(* Schneider Machine Expert - Basic project control, file version 2.9.0.0 *)
(* ProjectInformations: Name=Nuevo proyecto *)

HARDWARE
  Cpu 0: TM221M16R/G
  EthernetConfiguration: NetworkName=M221, IpAllocationMode=FixedAddress, IpAddress=0.0.0.0, SubnetMask=0.0.0.0
  SerialLineConfiguration: Baud=Baud19200, Parity=ParityEven, DataBits=DataBits8, StopBits=StopBits1, PhysicalMedium=PhysicalMediumRs485, TransmissionMode=TransmissionModeModbusRtu, SlaveId=1, Addressing=SlaveAddressing
  MastTask: UsePeriodScanMode=true, PeriodScan=10
  FastTask: Period=255
  CpuBehavior: StartingMode=StartAsPreviousState, AutoSaveRamOnEeprom=true, WatchdogPeriod=250

SYMBOLS  (address, symbol, comment, settings)
  %MW500    ERR
  %MW501    VEL
  %MW502    THETA
  %MW503    CRISP
  %MF1      REAL_ERROR
  %MF10     ENL
  %MF19     ENM
  %MF28     ENP
  %MF37     EZ
  %MF46     EPP
  %MF55     EPM
  %MF64     EPL
  %MF67     REAL_VEL
  %MF76     VNL
  %MF85     VNM
  %MF94     VNP
  %MF103    VZ
  %MF112    VPP
  %MF121    VPM
  %MF130    VPL
  %MF133    REAL_THETA
  %MF142    NL
  %MF151    NM
  %MF160    Z
  %MF169    PM
  %MF178    PL
  %MF181    W1
  %MF184    W2
  %MF187    W3
  %MF190    W4
  %MF193    W5
  %MF196    W6
  %MF199    W7
  %MF202    W8
  %MF205    W9
  %MF208    W10
  %MF211    W11
  %MF214    W12
  %MF217    W13
  %MF220    W14
  %MF223    W15
  %MF226    W16
  %MF229    W17
  %MF232    W18
  %MF235    W19
  %MF238    W20
  %MF241    W21
  %MF244    W22
  %MF247    W23
  %MF250    W24
  %MF253    W25
  %MF283    NUM
  %MF301    DEN

POU Nuevo POU
  (* SectionNumber=1 *)

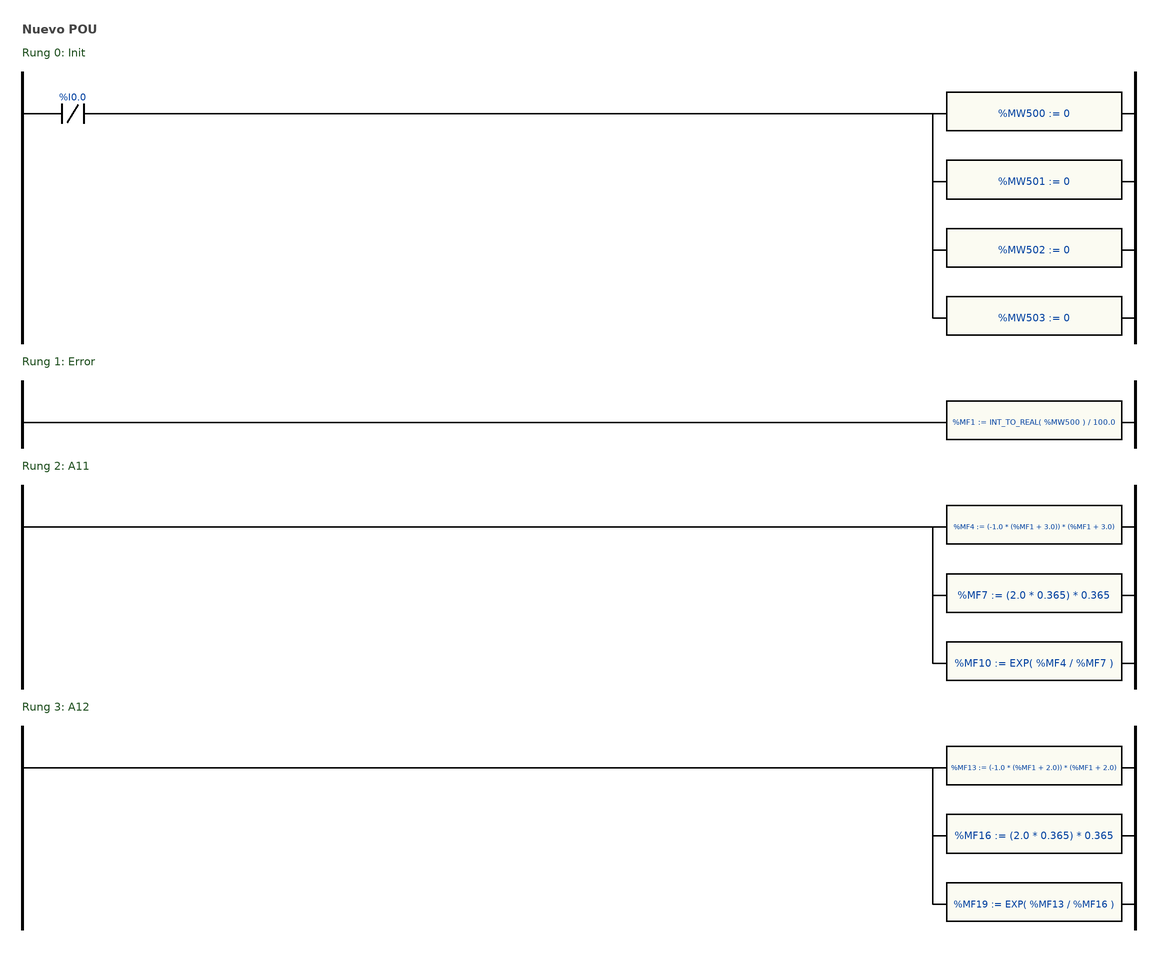

// Rung 0: Init
  LDN %I0.0
  [ %MW500 := 0 ]         (* ERR *)
  [ %MW501 := 0 ]         (* VEL *)
  [ %MW502 := 0 ]         (* THETA *)
  [ %MW503 := 0 ]         (* CRISP *)
  // as ST:
  //   IF NOT %I0.0 THEN ERR := 0; END_IF;
  //   IF NOT %I0.0 THEN VEL := 0; END_IF;
  //   IF NOT %I0.0 THEN THETA := 0; END_IF;
  //   IF NOT %I0.0 THEN CRISP := 0; END_IF;

// Rung 1: Error
  LD 1
  [ %MF1 := INT_TO_REAL ( %MW500 ) / 100.0 ](* REAL_ERROR, ERR *)
  // as ST:
  //   REAL_ERROR := INT_TO_REAL ( ERR ) / 100.0;

// Rung 2: A11
  LD 1
  [ %MF4 := ( -1.0 * ( %MF1 + 3.0 ) ) * ( %MF1 + 3.0 ) ](* REAL_ERROR, REAL_ERROR *)
  [ %MF7 := ( 2.0 * 0.365 ) * 0.365 ]
  [ %MF10 := EXP ( %MF4 / %MF7 ) ](* ENL *)
  // as ST:
  //   %MF4 := ( -1.0 * ( REAL_ERROR + 3.0 ) ) * ( REAL_ERROR + 3.0 );
  //   %MF7 := ( 2.0 * 0.365 ) * 0.365;
  //   ENL := EXP ( %MF4 / %MF7 );

// Rung 3: A12
  LD 1
  [ %MF13 := ( -1.0 * ( %MF1 + 2.0 ) ) * ( %MF1 + 2.0 ) ](* REAL_ERROR, REAL_ERROR *)
  [ %MF16 := ( 2.0 * 0.365 ) * 0.365 ]
  [ %MF19 := EXP ( %MF13 / %MF16 ) ](* ENM *)
  // as ST:
  //   %MF13 := ( -1.0 * ( REAL_ERROR + 2.0 ) ) * ( REAL_ERROR + 2.0 );
  //   %MF16 := ( 2.0 * 0.365 ) * 0.365;
  //   ENM := EXP ( %MF13 / %MF16 );

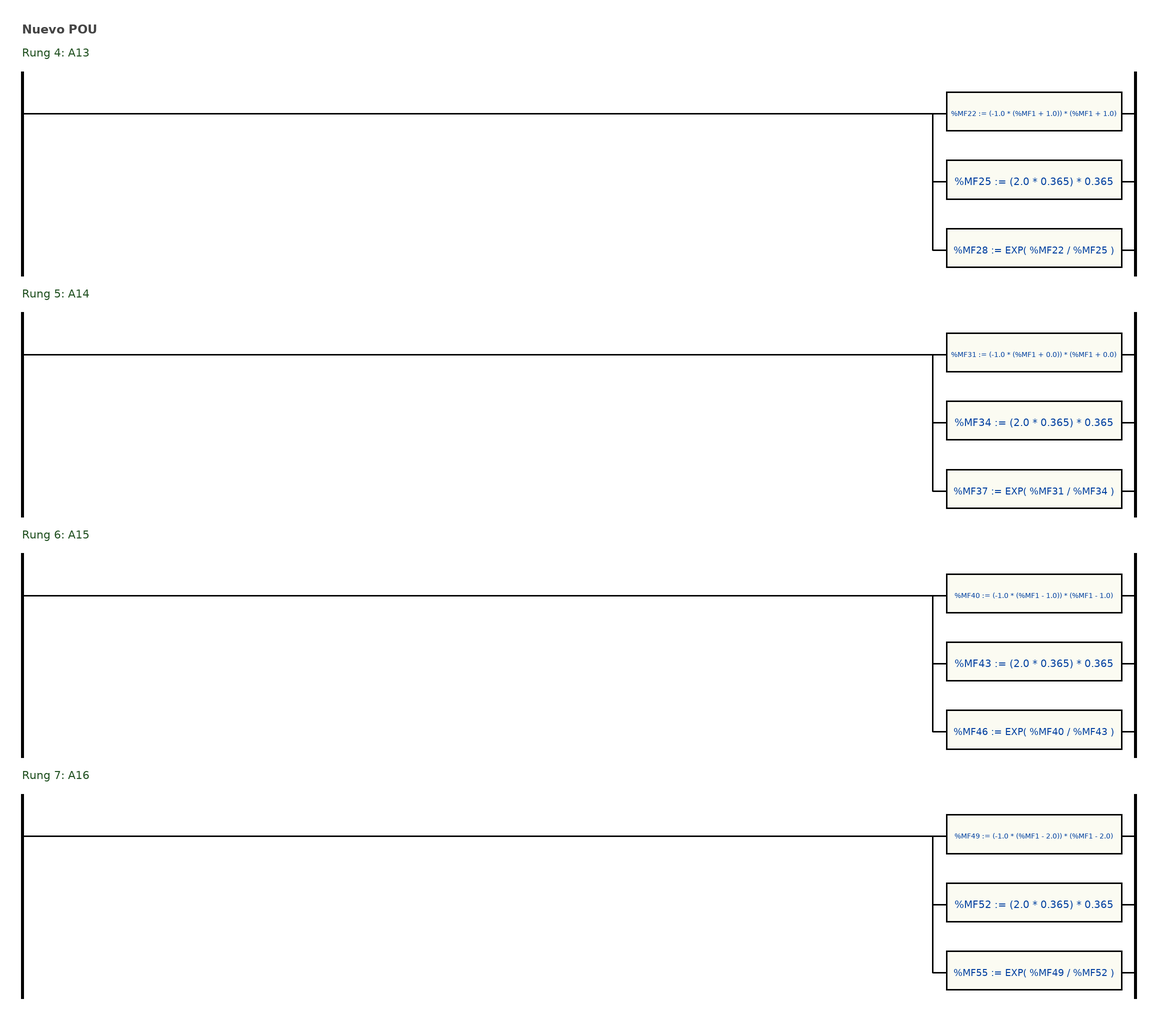

// Rung 4: A13
  LD 1
  [ %MF22 := ( -1.0 * ( %MF1 + 1.0 ) ) * ( %MF1 + 1.0 ) ](* REAL_ERROR, REAL_ERROR *)
  [ %MF25 := ( 2.0 * 0.365 ) * 0.365 ]
  [ %MF28 := EXP ( %MF22 / %MF25 ) ](* ENP *)
  // as ST:
  //   %MF22 := ( -1.0 * ( REAL_ERROR + 1.0 ) ) * ( REAL_ERROR + 1.0 );
  //   %MF25 := ( 2.0 * 0.365 ) * 0.365;
  //   ENP := EXP ( %MF22 / %MF25 );

// Rung 5: A14
  LD 1
  [ %MF31 := ( -1.0 * ( %MF1 + 0.0 ) ) * ( %MF1 + 0.0 ) ](* REAL_ERROR, REAL_ERROR *)
  [ %MF34 := ( 2.0 * 0.365 ) * 0.365 ]
  [ %MF37 := EXP ( %MF31 / %MF34 ) ](* EZ *)
  // as ST:
  //   %MF31 := ( -1.0 * ( REAL_ERROR + 0.0 ) ) * ( REAL_ERROR + 0.0 );
  //   %MF34 := ( 2.0 * 0.365 ) * 0.365;
  //   EZ := EXP ( %MF31 / %MF34 );

// Rung 6: A15
  LD 1
  [ %MF40 := ( -1.0 * ( %MF1 - 1.0 ) ) * ( %MF1 - 1.0 ) ](* REAL_ERROR, REAL_ERROR *)
  [ %MF43 := ( 2.0 * 0.365 ) * 0.365 ]
  [ %MF46 := EXP ( %MF40 / %MF43 ) ](* EPP *)
  // as ST:
  //   %MF40 := ( -1.0 * ( REAL_ERROR - 1.0 ) ) * ( REAL_ERROR - 1.0 );
  //   %MF43 := ( 2.0 * 0.365 ) * 0.365;
  //   EPP := EXP ( %MF40 / %MF43 );

// Rung 7: A16
  LD 1
  [ %MF49 := ( -1.0 * ( %MF1 - 2.0 ) ) * ( %MF1 - 2.0 ) ](* REAL_ERROR, REAL_ERROR *)
  [ %MF52 := ( 2.0 * 0.365 ) * 0.365 ]
  [ %MF55 := EXP ( %MF49 / %MF52 ) ](* EPM *)
  // as ST:
  //   %MF49 := ( -1.0 * ( REAL_ERROR - 2.0 ) ) * ( REAL_ERROR - 2.0 );
  //   %MF52 := ( 2.0 * 0.365 ) * 0.365;
  //   EPM := EXP ( %MF49 / %MF52 );

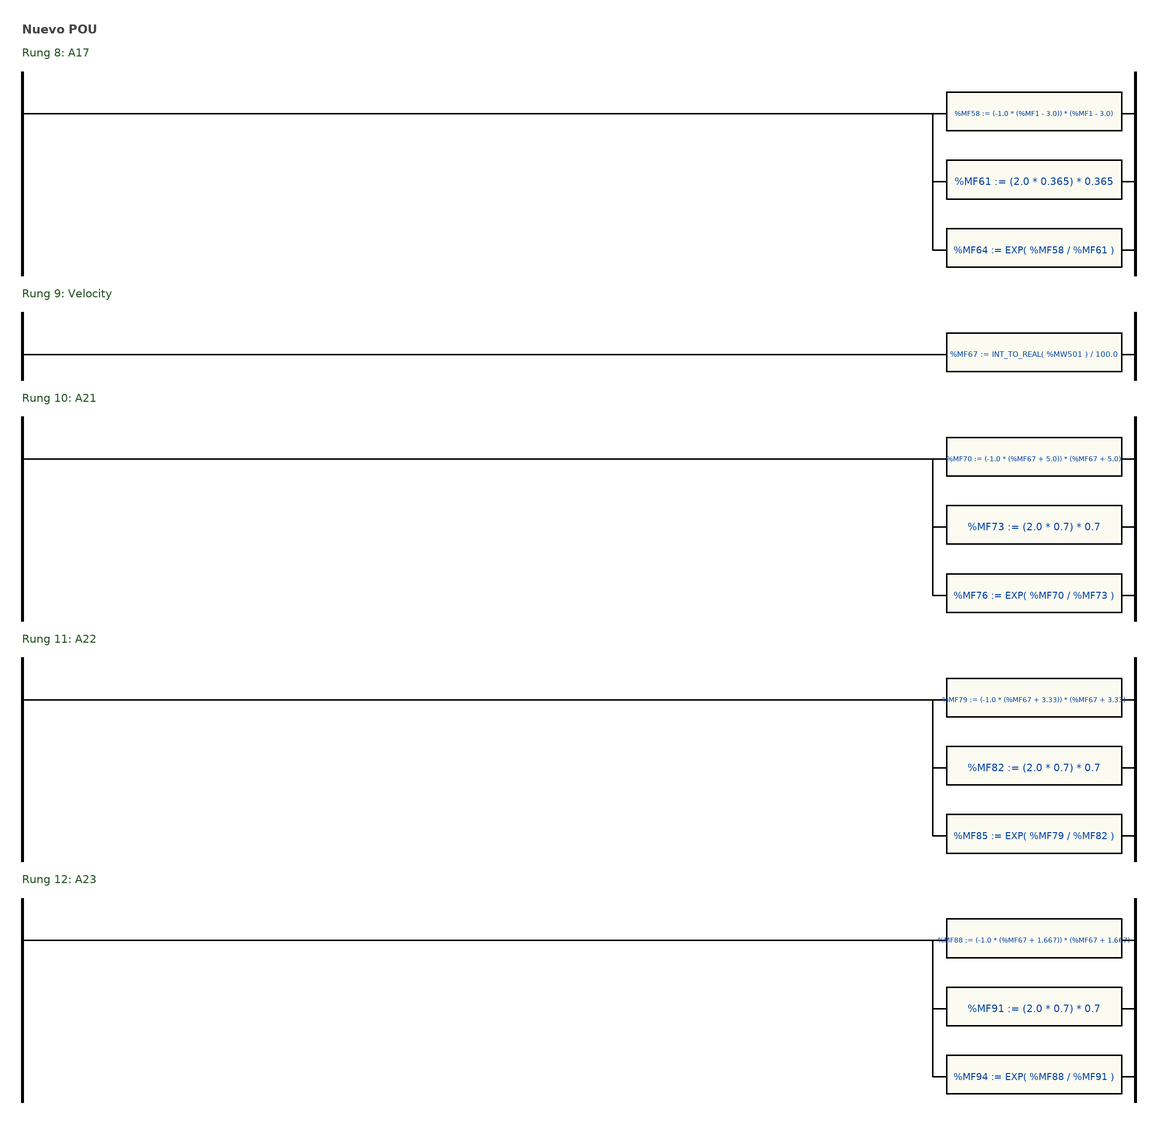

// Rung 8: A17
  LD 1
  [ %MF58 := ( -1.0 * ( %MF1 - 3.0 ) ) * ( %MF1 - 3.0 ) ](* REAL_ERROR, REAL_ERROR *)
  [ %MF61 := ( 2.0 * 0.365 ) * 0.365 ]
  [ %MF64 := EXP ( %MF58 / %MF61 ) ](* EPL *)
  // as ST:
  //   %MF58 := ( -1.0 * ( REAL_ERROR - 3.0 ) ) * ( REAL_ERROR - 3.0 );
  //   %MF61 := ( 2.0 * 0.365 ) * 0.365;
  //   EPL := EXP ( %MF58 / %MF61 );

// Rung 9: Velocity
  LD 1
  [ %MF67 := INT_TO_REAL ( %MW501 ) / 100.0 ](* REAL_VEL, VEL *)
  // as ST:
  //   REAL_VEL := INT_TO_REAL ( VEL ) / 100.0;

// Rung 10: A21
  LD 1
  [ %MF70 := ( -1.0 * ( %MF67 + 5.0 ) ) * ( %MF67 + 5.0 ) ](* REAL_VEL, REAL_VEL *)
  [ %MF73 := ( 2.0 * 0.7 ) * 0.7 ]
  [ %MF76 := EXP ( %MF70 / %MF73 ) ](* VNL *)
  // as ST:
  //   %MF70 := ( -1.0 * ( REAL_VEL + 5.0 ) ) * ( REAL_VEL + 5.0 );
  //   %MF73 := ( 2.0 * 0.7 ) * 0.7;
  //   VNL := EXP ( %MF70 / %MF73 );

// Rung 11: A22
  LD 1
  [ %MF79 := ( -1.0 * ( %MF67 + 3.33 ) ) * ( %MF67 + 3.33 ) ](* REAL_VEL, REAL_VEL *)
  [ %MF82 := ( 2.0 * 0.7 ) * 0.7 ]
  [ %MF85 := EXP ( %MF79 / %MF82 ) ](* VNM *)
  // as ST:
  //   %MF79 := ( -1.0 * ( REAL_VEL + 3.33 ) ) * ( REAL_VEL + 3.33 );
  //   %MF82 := ( 2.0 * 0.7 ) * 0.7;
  //   VNM := EXP ( %MF79 / %MF82 );

// Rung 12: A23
  LD 1
  [ %MF88 := ( -1.0 * ( %MF67 + 1.667 ) ) * ( %MF67 + 1.667 ) ](* REAL_VEL, REAL_VEL *)
  [ %MF91 := ( 2.0 * 0.7 ) * 0.7 ]
  [ %MF94 := EXP ( %MF88 / %MF91 ) ](* VNP *)
  // as ST:
  //   %MF88 := ( -1.0 * ( REAL_VEL + 1.667 ) ) * ( REAL_VEL + 1.667 );
  //   %MF91 := ( 2.0 * 0.7 ) * 0.7;
  //   VNP := EXP ( %MF88 / %MF91 );

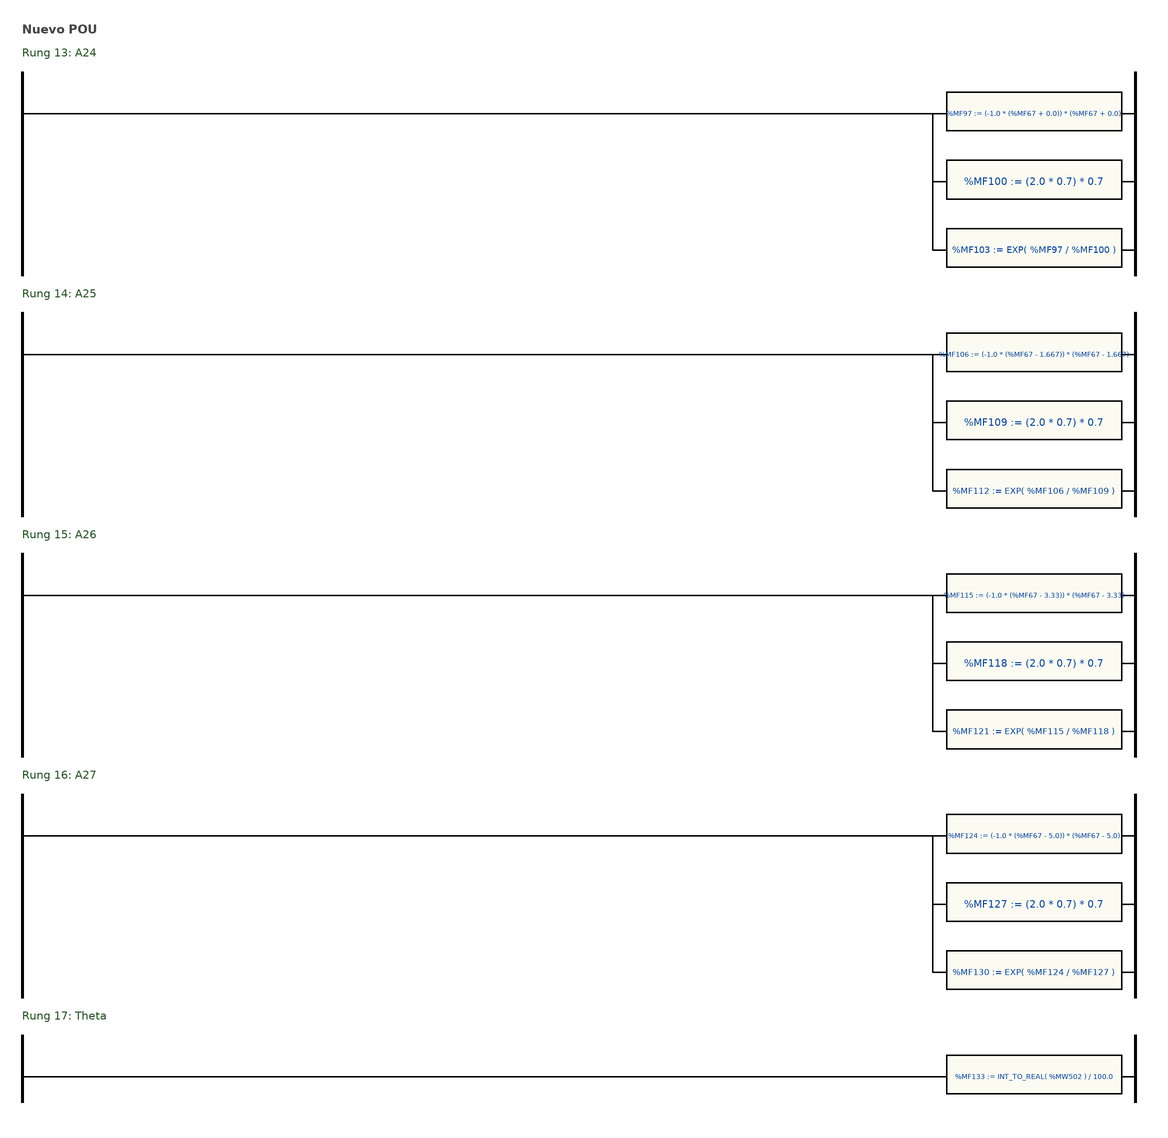

// Rung 13: A24
  LD 1
  [ %MF97 := ( -1.0 * ( %MF67 + 0.0 ) ) * ( %MF67 + 0.0 ) ](* REAL_VEL, REAL_VEL *)
  [ %MF100 := ( 2.0 * 0.7 ) * 0.7 ]
  [ %MF103 := EXP ( %MF97 / %MF100 ) ](* VZ *)
  // as ST:
  //   %MF97 := ( -1.0 * ( REAL_VEL + 0.0 ) ) * ( REAL_VEL + 0.0 );
  //   %MF100 := ( 2.0 * 0.7 ) * 0.7;
  //   VZ := EXP ( %MF97 / %MF100 );

// Rung 14: A25
  LD 1
  [ %MF106 := ( -1.0 * ( %MF67 - 1.667 ) ) * ( %MF67 - 1.667 ) ](* REAL_VEL, REAL_VEL *)
  [ %MF109 := ( 2.0 * 0.7 ) * 0.7 ]
  [ %MF112 := EXP ( %MF106 / %MF109 ) ](* VPP *)
  // as ST:
  //   %MF106 := ( -1.0 * ( REAL_VEL - 1.667 ) ) * ( REAL_VEL - 1.667 );
  //   %MF109 := ( 2.0 * 0.7 ) * 0.7;
  //   VPP := EXP ( %MF106 / %MF109 );

// Rung 15: A26
  LD 1
  [ %MF115 := ( -1.0 * ( %MF67 - 3.33 ) ) * ( %MF67 - 3.33 ) ](* REAL_VEL, REAL_VEL *)
  [ %MF118 := ( 2.0 * 0.7 ) * 0.7 ]
  [ %MF121 := EXP ( %MF115 / %MF118 ) ](* VPM *)
  // as ST:
  //   %MF115 := ( -1.0 * ( REAL_VEL - 3.33 ) ) * ( REAL_VEL - 3.33 );
  //   %MF118 := ( 2.0 * 0.7 ) * 0.7;
  //   VPM := EXP ( %MF115 / %MF118 );

// Rung 16: A27
  LD 1
  [ %MF124 := ( -1.0 * ( %MF67 - 5.0 ) ) * ( %MF67 - 5.0 ) ](* REAL_VEL, REAL_VEL *)
  [ %MF127 := ( 2.0 * 0.7 ) * 0.7 ]
  [ %MF130 := EXP ( %MF124 / %MF127 ) ](* VPL *)
  // as ST:
  //   %MF124 := ( -1.0 * ( REAL_VEL - 5.0 ) ) * ( REAL_VEL - 5.0 );
  //   %MF127 := ( 2.0 * 0.7 ) * 0.7;
  //   VPL := EXP ( %MF124 / %MF127 );

// Rung 17: Theta
  LD 1
  [ %MF133 := INT_TO_REAL ( %MW502 ) / 100.0 ](* REAL_THETA, THETA *)
  // as ST:
  //   REAL_THETA := INT_TO_REAL ( THETA ) / 100.0;

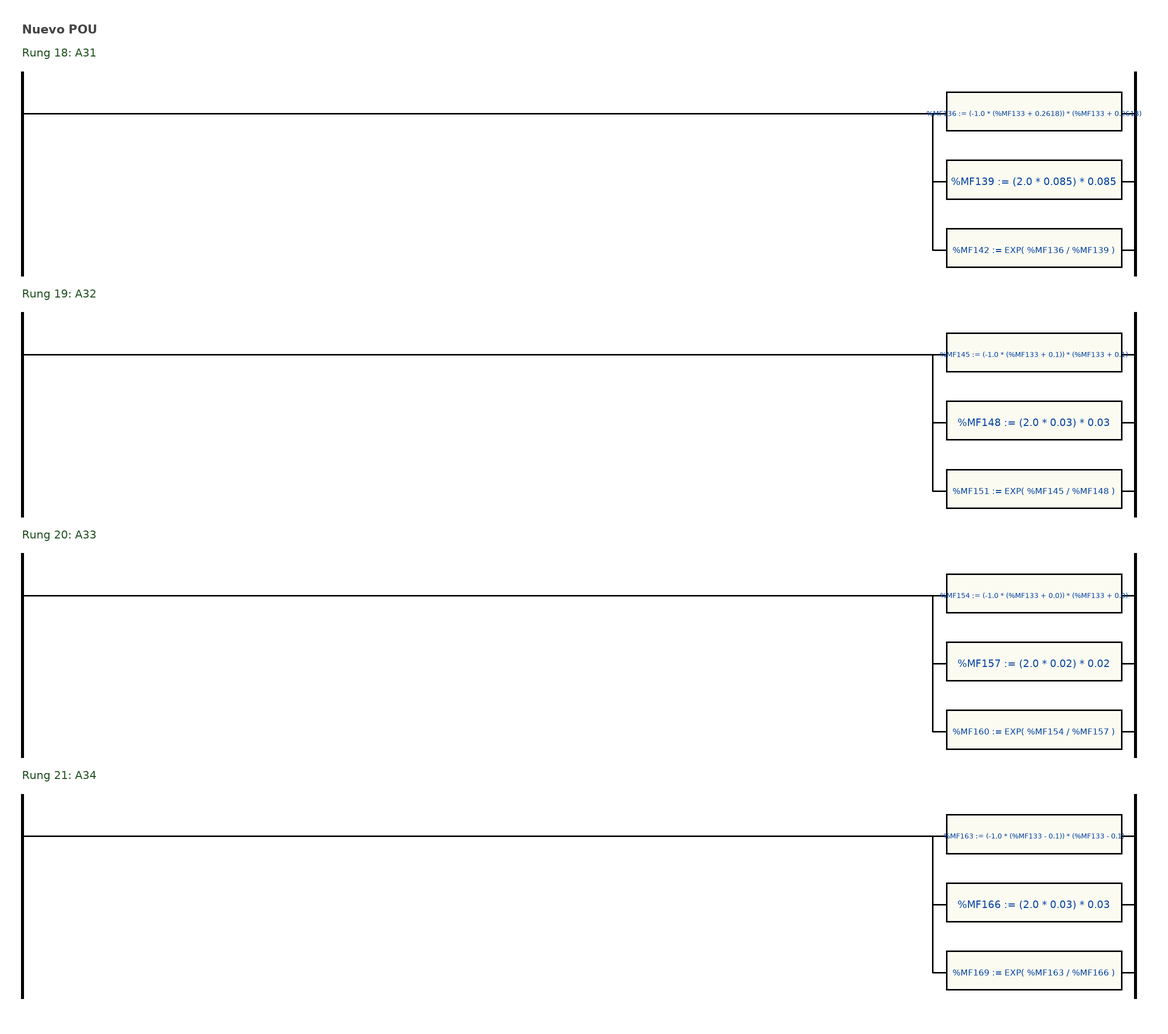

// Rung 18: A31
  LD 1
  [ %MF136 := ( -1.0 * ( %MF133 + 0.2618 ) ) * ( %MF133 + 0.2618 ) ](* REAL_THETA, REAL_THETA *)
  [ %MF139 := ( 2.0 * 0.085 ) * 0.085 ]
  [ %MF142 := EXP ( %MF136 / %MF139 ) ](* NL *)
  // as ST:
  //   %MF136 := ( -1.0 * ( REAL_THETA + 0.2618 ) ) * ( REAL_THETA + 0.2618 );
  //   %MF139 := ( 2.0 * 0.085 ) * 0.085;
  //   NL := EXP ( %MF136 / %MF139 );

// Rung 19: A32
  LD 1
  [ %MF145 := ( -1.0 * ( %MF133 + 0.1 ) ) * ( %MF133 + 0.1 ) ](* REAL_THETA, REAL_THETA *)
  [ %MF148 := ( 2.0 * 0.03 ) * 0.03 ]
  [ %MF151 := EXP ( %MF145 / %MF148 ) ](* NM *)
  // as ST:
  //   %MF145 := ( -1.0 * ( REAL_THETA + 0.1 ) ) * ( REAL_THETA + 0.1 );
  //   %MF148 := ( 2.0 * 0.03 ) * 0.03;
  //   NM := EXP ( %MF145 / %MF148 );

// Rung 20: A33
  LD 1
  [ %MF154 := ( -1.0 * ( %MF133 + 0.0 ) ) * ( %MF133 + 0.0 ) ](* REAL_THETA, REAL_THETA *)
  [ %MF157 := ( 2.0 * 0.02 ) * 0.02 ]
  [ %MF160 := EXP ( %MF154 / %MF157 ) ](* Z *)
  // as ST:
  //   %MF154 := ( -1.0 * ( REAL_THETA + 0.0 ) ) * ( REAL_THETA + 0.0 );
  //   %MF157 := ( 2.0 * 0.02 ) * 0.02;
  //   Z := EXP ( %MF154 / %MF157 );

// Rung 21: A34
  LD 1
  [ %MF163 := ( -1.0 * ( %MF133 - 0.1 ) ) * ( %MF133 - 0.1 ) ](* REAL_THETA, REAL_THETA *)
  [ %MF166 := ( 2.0 * 0.03 ) * 0.03 ]
  [ %MF169 := EXP ( %MF163 / %MF166 ) ](* PM *)
  // as ST:
  //   %MF163 := ( -1.0 * ( REAL_THETA - 0.1 ) ) * ( REAL_THETA - 0.1 );
  //   %MF166 := ( 2.0 * 0.03 ) * 0.03;
  //   PM := EXP ( %MF163 / %MF166 );

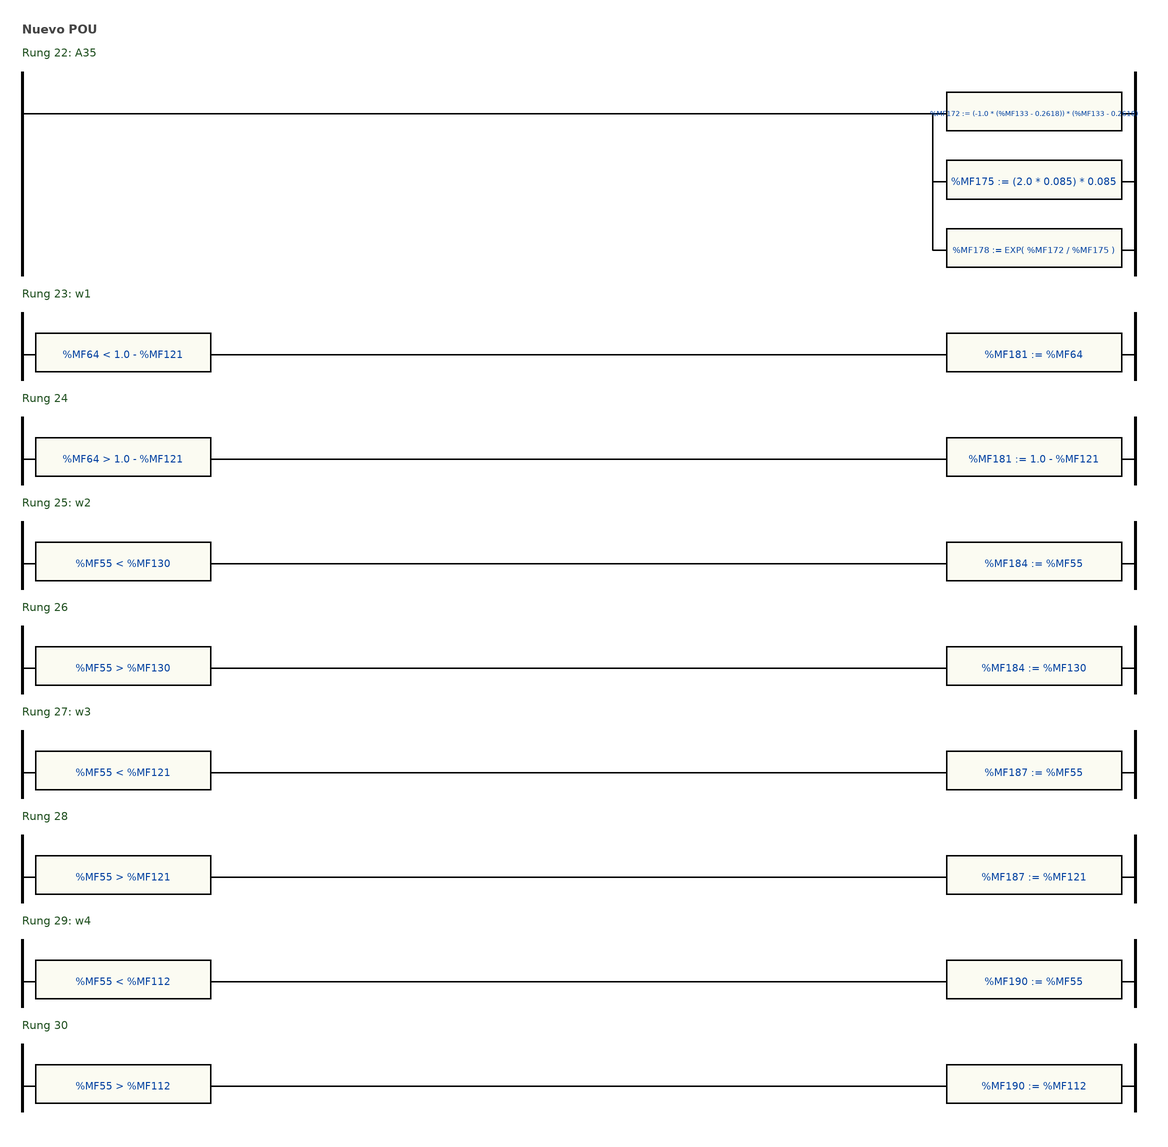

// Rung 22: A35
  LD 1
  [ %MF172 := ( -1.0 * ( %MF133 - 0.2618 ) ) * ( %MF133 - 0.2618 ) ](* REAL_THETA, REAL_THETA *)
  [ %MF175 := ( 2.0 * 0.085 ) * 0.085 ]
  [ %MF178 := EXP ( %MF172 / %MF175 ) ](* PL *)
  // as ST:
  //   %MF172 := ( -1.0 * ( REAL_THETA - 0.2618 ) ) * ( REAL_THETA - 0.2618 );
  //   %MF175 := ( 2.0 * 0.085 ) * 0.085;
  //   PL := EXP ( %MF172 / %MF175 );

// Rung 23: w1
  LD 1
  AND [ %MF64 < 1.0 - %MF121 ](* EPL, VPM *)
  [ %MF181 := %MF64 ]     (* W1, EPL *)
  // as ST:
  //   IF EPL < 1.0 - VPM THEN W1 := EPL; END_IF;

// Rung 24
  LD 1
  AND [ %MF64 > 1.0 - %MF121 ](* EPL, VPM *)
  [ %MF181 := 1.0 - %MF121 ](* W1, VPM *)
  // as ST:
  //   IF EPL > 1.0 - VPM THEN W1 := 1.0 - VPM; END_IF;

// Rung 25: w2
  LD [ %MF55 < %MF130 ]   (* EPM, VPL *)
  [ %MF184 := %MF55 ]     (* W2, EPM *)
  // as ST:
  //   IF EPM < VPL THEN W2 := EPM; END_IF;

// Rung 26
  LD [ %MF55 > %MF130 ]   (* EPM, VPL *)
  [ %MF184 := %MF130 ]    (* W2, VPL *)
  // as ST:
  //   IF EPM > VPL THEN W2 := VPL; END_IF;

// Rung 27: w3
  LD [ %MF55 < %MF121 ]   (* EPM, VPM *)
  [ %MF187 := %MF55 ]     (* W3, EPM *)
  // as ST:
  //   IF EPM < VPM THEN W3 := EPM; END_IF;

// Rung 28
  LD [ %MF55 > %MF121 ]   (* EPM, VPM *)
  [ %MF187 := %MF121 ]    (* W3, VPM *)
  // as ST:
  //   IF EPM > VPM THEN W3 := VPM; END_IF;

// Rung 29: w4
  LD [ %MF55 < %MF112 ]   (* EPM, VPP *)
  [ %MF190 := %MF55 ]     (* W4, EPM *)
  // as ST:
  //   IF EPM < VPP THEN W4 := EPM; END_IF;

// Rung 30
  LD [ %MF55 > %MF112 ]   (* EPM, VPP *)
  [ %MF190 := %MF112 ]    (* W4, VPP *)
  // as ST:
  //   IF EPM > VPP THEN W4 := VPP; END_IF;

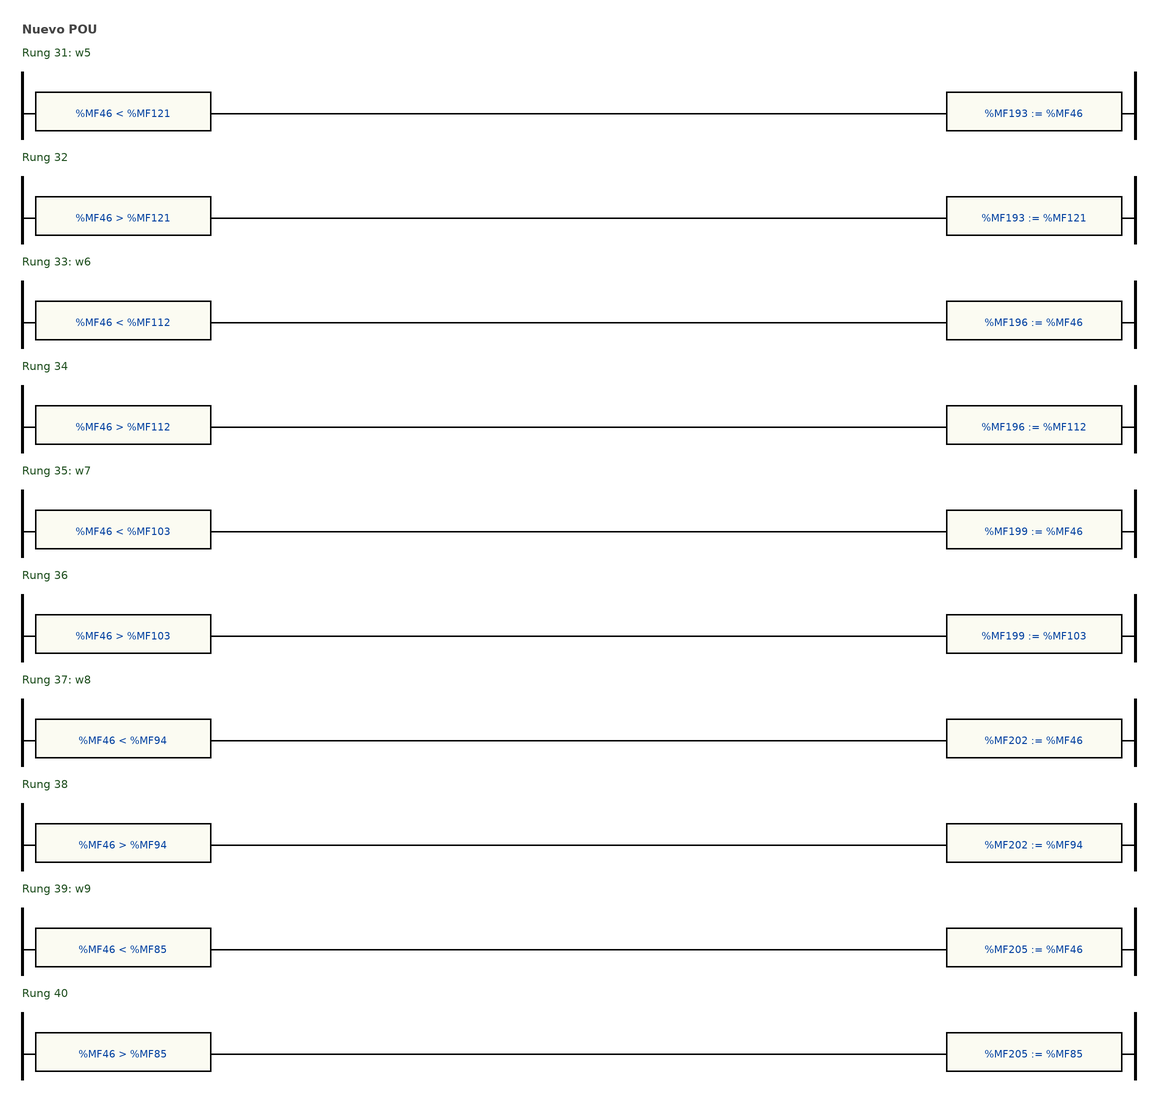

// Rung 31: w5
  LD [ %MF46 < %MF121 ]   (* EPP, VPM *)
  [ %MF193 := %MF46 ]     (* W5, EPP *)
  // as ST:
  //   IF EPP < VPM THEN W5 := EPP; END_IF;

// Rung 32
  LD [ %MF46 > %MF121 ]   (* EPP, VPM *)
  [ %MF193 := %MF121 ]    (* W5, VPM *)
  // as ST:
  //   IF EPP > VPM THEN W5 := VPM; END_IF;

// Rung 33: w6
  LD [ %MF46 < %MF112 ]   (* EPP, VPP *)
  [ %MF196 := %MF46 ]     (* W6, EPP *)
  // as ST:
  //   IF EPP < VPP THEN W6 := EPP; END_IF;

// Rung 34
  LD [ %MF46 > %MF112 ]   (* EPP, VPP *)
  [ %MF196 := %MF112 ]    (* W6, VPP *)
  // as ST:
  //   IF EPP > VPP THEN W6 := VPP; END_IF;

// Rung 35: w7
  LD [ %MF46 < %MF103 ]   (* EPP, VZ *)
  [ %MF199 := %MF46 ]     (* W7, EPP *)
  // as ST:
  //   IF EPP < VZ THEN W7 := EPP; END_IF;

// Rung 36
  LD [ %MF46 > %MF103 ]   (* EPP, VZ *)
  [ %MF199 := %MF103 ]    (* W7, VZ *)
  // as ST:
  //   IF EPP > VZ THEN W7 := VZ; END_IF;

// Rung 37: w8
  LD [ %MF46 < %MF94 ]    (* EPP, VNP *)
  [ %MF202 := %MF46 ]     (* W8, EPP *)
  // as ST:
  //   IF EPP < VNP THEN W8 := EPP; END_IF;

// Rung 38
  LD [ %MF46 > %MF94 ]    (* EPP, VNP *)
  [ %MF202 := %MF94 ]     (* W8, VNP *)
  // as ST:
  //   IF EPP > VNP THEN W8 := VNP; END_IF;

// Rung 39: w9
  LD [ %MF46 < %MF85 ]    (* EPP, VNM *)
  [ %MF205 := %MF46 ]     (* W9, EPP *)
  // as ST:
  //   IF EPP < VNM THEN W9 := EPP; END_IF;

// Rung 40
  LD [ %MF46 > %MF85 ]    (* EPP, VNM *)
  [ %MF205 := %MF85 ]     (* W9, VNM *)
  // as ST:
  //   IF EPP > VNM THEN W9 := VNM; END_IF;

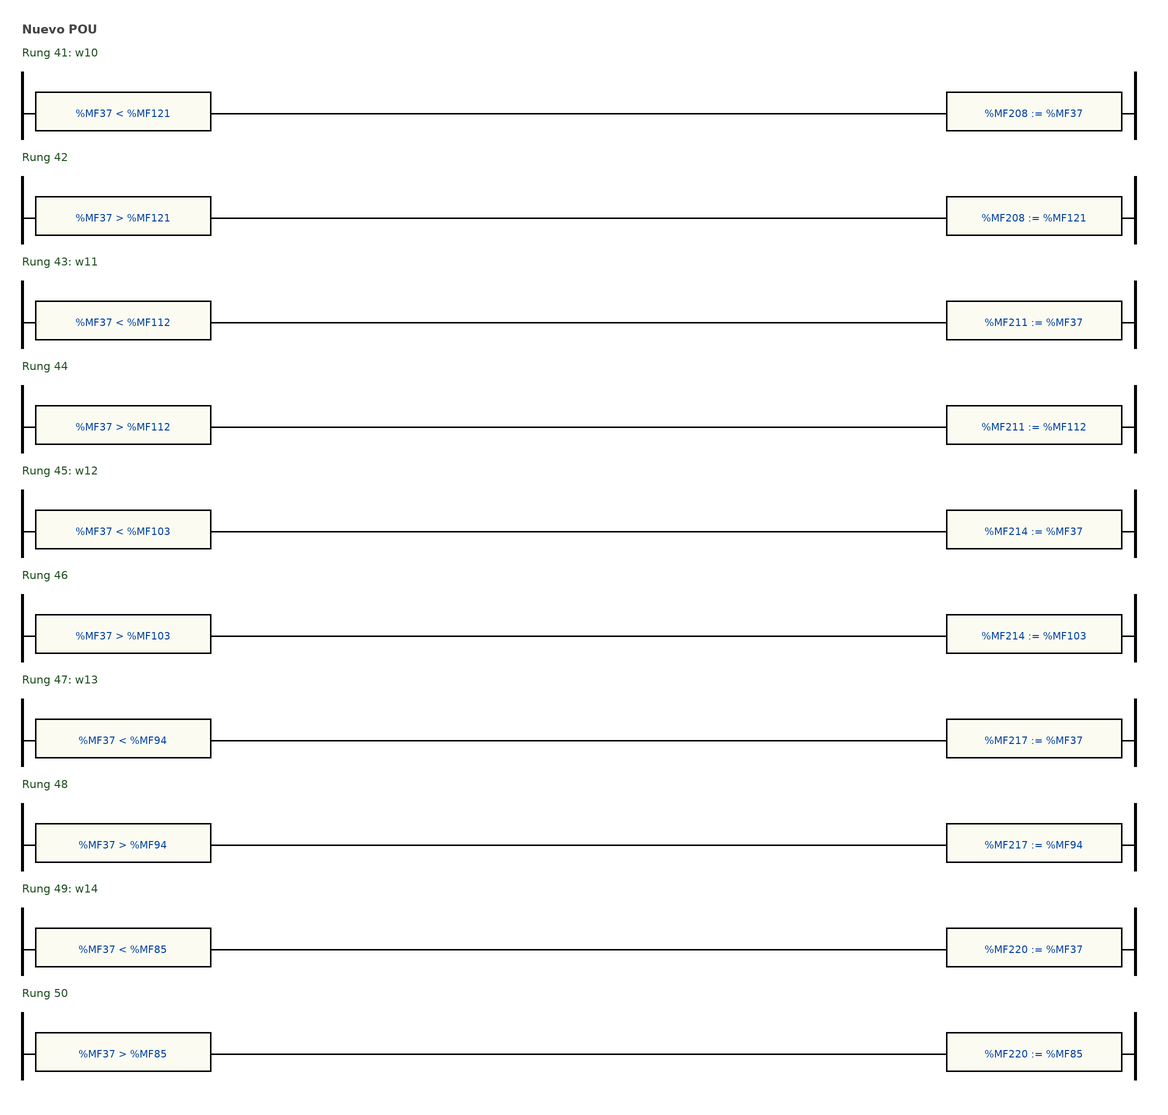

// Rung 41: w10
  LD [ %MF37 < %MF121 ]   (* EZ, VPM *)
  [ %MF208 := %MF37 ]     (* W10, EZ *)
  // as ST:
  //   IF EZ < VPM THEN W10 := EZ; END_IF;

// Rung 42
  LD [ %MF37 > %MF121 ]   (* EZ, VPM *)
  [ %MF208 := %MF121 ]    (* W10, VPM *)
  // as ST:
  //   IF EZ > VPM THEN W10 := VPM; END_IF;

// Rung 43: w11
  LD [ %MF37 < %MF112 ]   (* EZ, VPP *)
  [ %MF211 := %MF37 ]     (* W11, EZ *)
  // as ST:
  //   IF EZ < VPP THEN W11 := EZ; END_IF;

// Rung 44
  LD [ %MF37 > %MF112 ]   (* EZ, VPP *)
  [ %MF211 := %MF112 ]    (* W11, VPP *)
  // as ST:
  //   IF EZ > VPP THEN W11 := VPP; END_IF;

// Rung 45: w12
  LD [ %MF37 < %MF103 ]   (* EZ, VZ *)
  [ %MF214 := %MF37 ]     (* W12, EZ *)
  // as ST:
  //   IF EZ < VZ THEN W12 := EZ; END_IF;

// Rung 46
  LD [ %MF37 > %MF103 ]   (* EZ, VZ *)
  [ %MF214 := %MF103 ]    (* W12, VZ *)
  // as ST:
  //   IF EZ > VZ THEN W12 := VZ; END_IF;

// Rung 47: w13
  LD [ %MF37 < %MF94 ]    (* EZ, VNP *)
  [ %MF217 := %MF37 ]     (* W13, EZ *)
  // as ST:
  //   IF EZ < VNP THEN W13 := EZ; END_IF;

// Rung 48
  LD [ %MF37 > %MF94 ]    (* EZ, VNP *)
  [ %MF217 := %MF94 ]     (* W13, VNP *)
  // as ST:
  //   IF EZ > VNP THEN W13 := VNP; END_IF;

// Rung 49: w14
  LD [ %MF37 < %MF85 ]    (* EZ, VNM *)
  [ %MF220 := %MF37 ]     (* W14, EZ *)
  // as ST:
  //   IF EZ < VNM THEN W14 := EZ; END_IF;

// Rung 50
  LD [ %MF37 > %MF85 ]    (* EZ, VNM *)
  [ %MF220 := %MF85 ]     (* W14, VNM *)
  // as ST:
  //   IF EZ > VNM THEN W14 := VNM; END_IF;

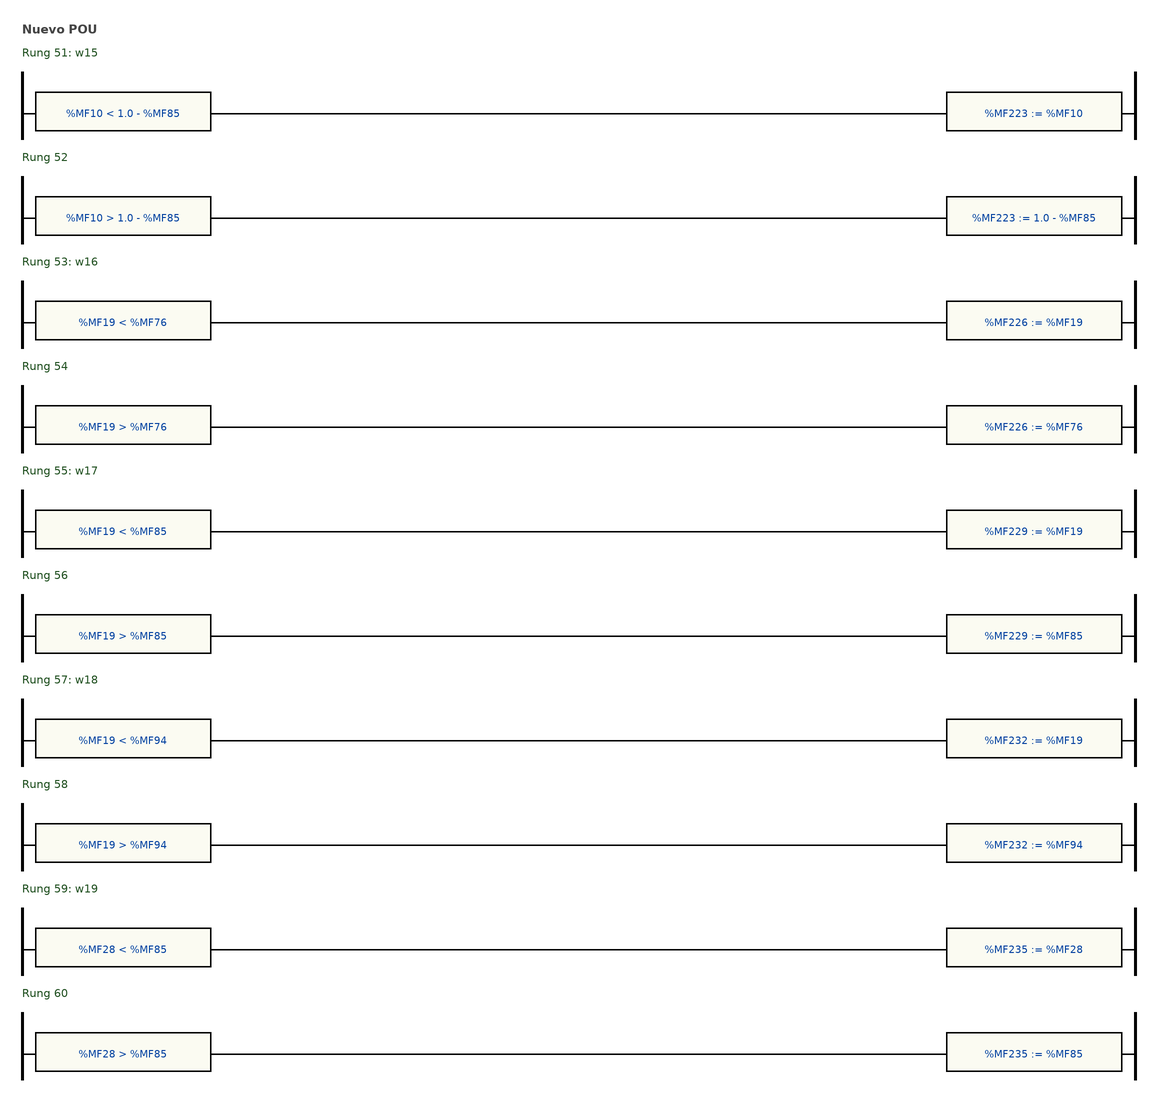

// Rung 51: w15
  LD 1
  AND [ %MF10 < 1.0 - %MF85 ](* ENL, VNM *)
  [ %MF223 := %MF10 ]     (* W15, ENL *)
  // as ST:
  //   IF ENL < 1.0 - VNM THEN W15 := ENL; END_IF;

// Rung 52
  LD 1
  AND [ %MF10 > 1.0 - %MF85 ](* ENL, VNM *)
  [ %MF223 := 1.0 - %MF85 ](* W15, VNM *)
  // as ST:
  //   IF ENL > 1.0 - VNM THEN W15 := 1.0 - VNM; END_IF;

// Rung 53: w16
  LD [ %MF19 < %MF76 ]    (* ENM, VNL *)
  [ %MF226 := %MF19 ]     (* W16, ENM *)
  // as ST:
  //   IF ENM < VNL THEN W16 := ENM; END_IF;

// Rung 54
  LD [ %MF19 > %MF76 ]    (* ENM, VNL *)
  [ %MF226 := %MF76 ]     (* W16, VNL *)
  // as ST:
  //   IF ENM > VNL THEN W16 := VNL; END_IF;

// Rung 55: w17
  LD [ %MF19 < %MF85 ]    (* ENM, VNM *)
  [ %MF229 := %MF19 ]     (* W17, ENM *)
  // as ST:
  //   IF ENM < VNM THEN W17 := ENM; END_IF;

// Rung 56
  LD [ %MF19 > %MF85 ]    (* ENM, VNM *)
  [ %MF229 := %MF85 ]     (* W17, VNM *)
  // as ST:
  //   IF ENM > VNM THEN W17 := VNM; END_IF;

// Rung 57: w18
  LD [ %MF19 < %MF94 ]    (* ENM, VNP *)
  [ %MF232 := %MF19 ]     (* W18, ENM *)
  // as ST:
  //   IF ENM < VNP THEN W18 := ENM; END_IF;

// Rung 58
  LD [ %MF19 > %MF94 ]    (* ENM, VNP *)
  [ %MF232 := %MF94 ]     (* W18, VNP *)
  // as ST:
  //   IF ENM > VNP THEN W18 := VNP; END_IF;

// Rung 59: w19
  LD [ %MF28 < %MF85 ]    (* ENP, VNM *)
  [ %MF235 := %MF28 ]     (* W19, ENP *)
  // as ST:
  //   IF ENP < VNM THEN W19 := ENP; END_IF;

// Rung 60
  LD [ %MF28 > %MF85 ]    (* ENP, VNM *)
  [ %MF235 := %MF85 ]     (* W19, VNM *)
  // as ST:
  //   IF ENP > VNM THEN W19 := VNM; END_IF;

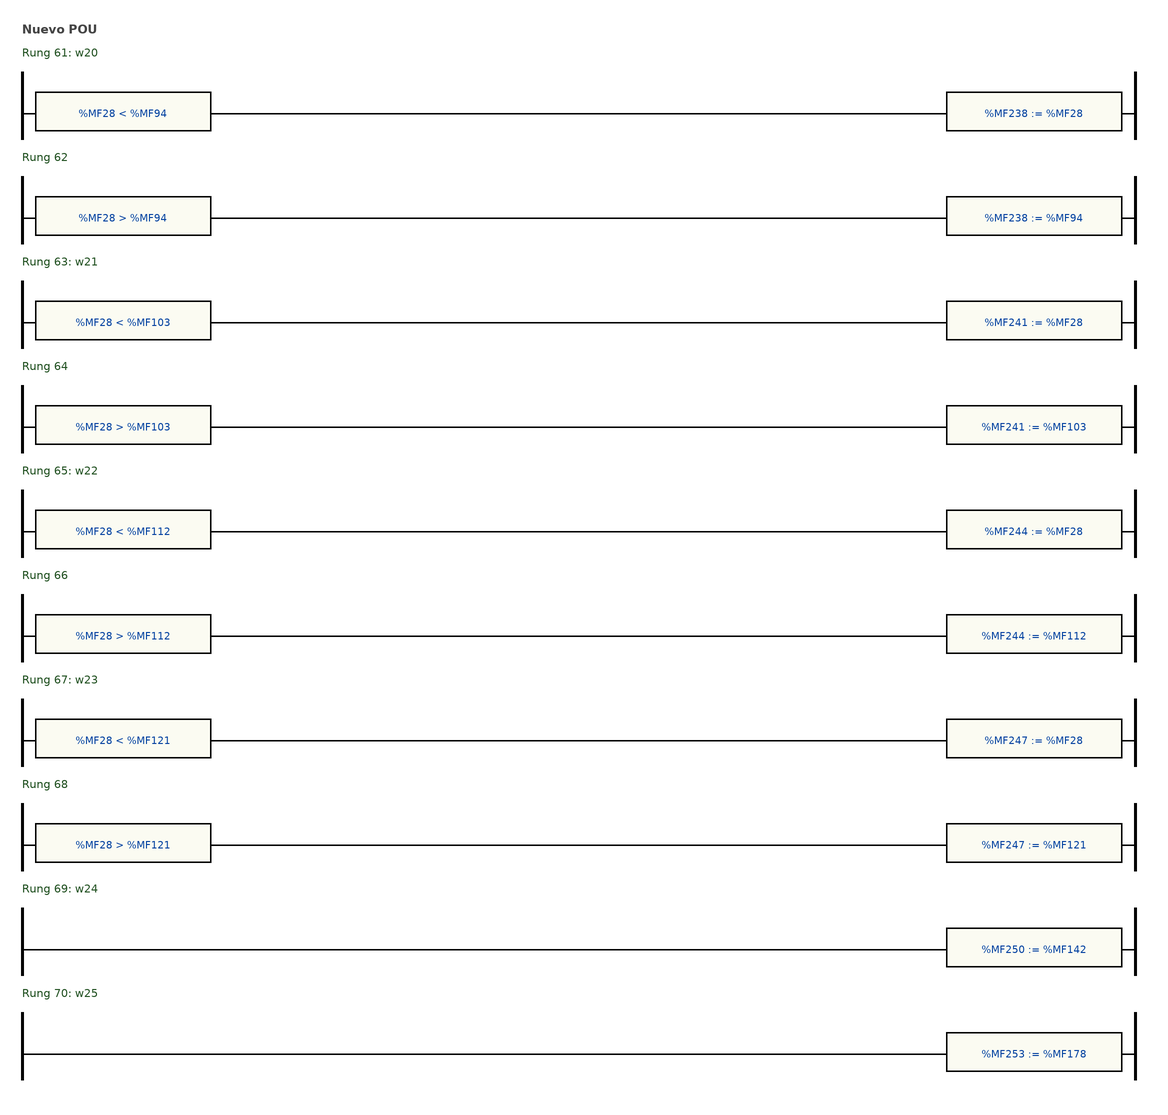

// Rung 61: w20
  LD [ %MF28 < %MF94 ]    (* ENP, VNP *)
  [ %MF238 := %MF28 ]     (* W20, ENP *)
  // as ST:
  //   IF ENP < VNP THEN W20 := ENP; END_IF;

// Rung 62
  LD [ %MF28 > %MF94 ]    (* ENP, VNP *)
  [ %MF238 := %MF94 ]     (* W20, VNP *)
  // as ST:
  //   IF ENP > VNP THEN W20 := VNP; END_IF;

// Rung 63: w21
  LD [ %MF28 < %MF103 ]   (* ENP, VZ *)
  [ %MF241 := %MF28 ]     (* W21, ENP *)
  // as ST:
  //   IF ENP < VZ THEN W21 := ENP; END_IF;

// Rung 64
  LD [ %MF28 > %MF103 ]   (* ENP, VZ *)
  [ %MF241 := %MF103 ]    (* W21, VZ *)
  // as ST:
  //   IF ENP > VZ THEN W21 := VZ; END_IF;

// Rung 65: w22
  LD [ %MF28 < %MF112 ]   (* ENP, VPP *)
  [ %MF244 := %MF28 ]     (* W22, ENP *)
  // as ST:
  //   IF ENP < VPP THEN W22 := ENP; END_IF;

// Rung 66
  LD [ %MF28 > %MF112 ]   (* ENP, VPP *)
  [ %MF244 := %MF112 ]    (* W22, VPP *)
  // as ST:
  //   IF ENP > VPP THEN W22 := VPP; END_IF;

// Rung 67: w23
  LD [ %MF28 < %MF121 ]   (* ENP, VPM *)
  [ %MF247 := %MF28 ]     (* W23, ENP *)
  // as ST:
  //   IF ENP < VPM THEN W23 := ENP; END_IF;

// Rung 68
  LD [ %MF28 > %MF121 ]   (* ENP, VPM *)
  [ %MF247 := %MF121 ]    (* W23, VPM *)
  // as ST:
  //   IF ENP > VPM THEN W23 := VPM; END_IF;

// Rung 69: w24
  LD 1
  [ %MF250 := %MF142 ]    (* W24, NL *)
  // as ST:
  //   W24 := NL;

// Rung 70: w25
  LD 1
  [ %MF253 := %MF178 ]    (* W25, PL *)
  // as ST:
  //   W25 := PL;

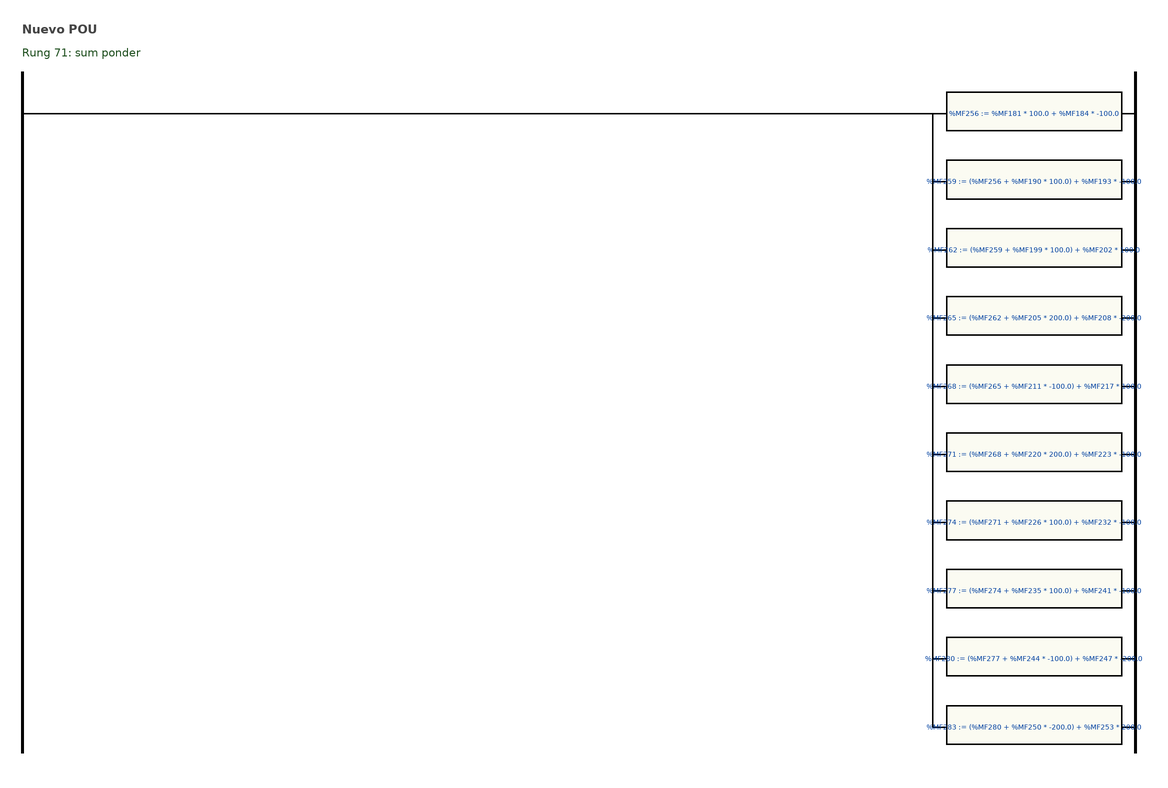

// Rung 71: sum ponder
  LD 1
  [ %MF256 := %MF181 * 100.0 + %MF184 * -100.0 ](* W1, W2 *)
  [ %MF259 := ( %MF256 + %MF190 * 100.0 ) + %MF193 * -100.0 ](* W4, W5 *)
  [ %MF262 := ( %MF259 + %MF199 * 100.0 ) + %MF202 * 100.0 ](* W7, W8 *)
  [ %MF265 := ( %MF262 + %MF205 * 200.0 ) + %MF208 * -200.0 ](* W9, W10 *)
  [ %MF268 := ( %MF265 + %MF211 * -100.0 ) + %MF217 * 100.0 ](* W11, W13 *)
  [ %MF271 := ( %MF268 + %MF220 * 200.0 ) + %MF223 * -100.0 ](* W14, W15 *)
  [ %MF274 := ( %MF271 + %MF226 * 100.0 ) + %MF232 * -100.0 ](* W16, W18 *)
  [ %MF277 := ( %MF274 + %MF235 * 100.0 ) + %MF241 * -100.0 ](* W19, W21 *)
  [ %MF280 := ( %MF277 + %MF244 * -100.0 ) + %MF247 * -200.0 ](* W22, W23 *)
  [ %MF283 := ( %MF280 + %MF250 * -200.0 ) + %MF253 * 200.0 ](* NUM, W24, W25 *)
  // as ST:
  //   %MF256 := W1 * 100.0 + W2 * -100.0;
  //   %MF259 := ( %MF256 + W4 * 100.0 ) + W5 * -100.0;
  //   %MF262 := ( %MF259 + W7 * 100.0 ) + W8 * 100.0;
  //   %MF265 := ( %MF262 + W9 * 200.0 ) + W10 * -200.0;
  //   %MF268 := ( %MF265 + W11 * -100.0 ) + W13 * 100.0;
  //   %MF271 := ( %MF268 + W14 * 200.0 ) + W15 * -100.0;
  //   %MF274 := ( %MF271 + W16 * 100.0 ) + W18 * -100.0;
  //   %MF277 := ( %MF274 + W19 * 100.0 ) + W21 * -100.0;
  //   %MF280 := ( %MF277 + W22 * -100.0 ) + W23 * -200.0;
  //   NUM := ( %MF280 + W24 * -200.0 ) + W25 * 200.0;

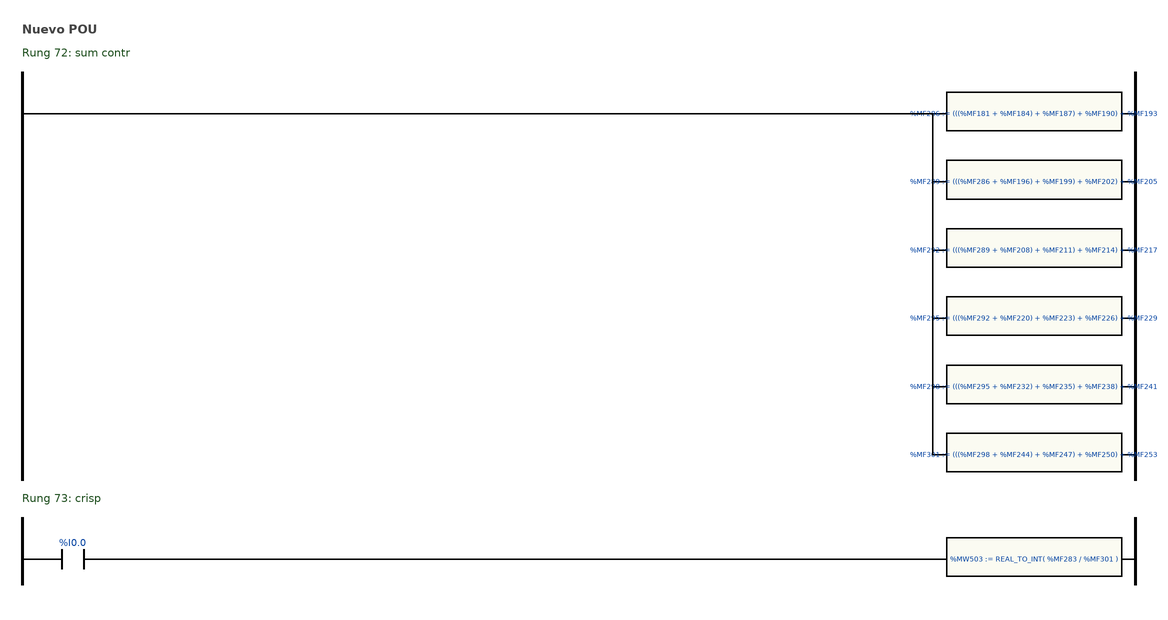

// Rung 72: sum contr
  LD 1
  [ %MF286 := ( ( ( %MF181 + %MF184 ) + %MF187 ) + %MF190 ) + %MF193 ](* W1, W2, W3, W4, W5 *)
  [ %MF289 := ( ( ( %MF286 + %MF196 ) + %MF199 ) + %MF202 ) + %MF205 ](* W6, W7, W8, W9 *)
  [ %MF292 := ( ( ( %MF289 + %MF208 ) + %MF211 ) + %MF214 ) + %MF217 ](* W10, W11, W12, W13 *)
  [ %MF295 := ( ( ( %MF292 + %MF220 ) + %MF223 ) + %MF226 ) + %MF229 ](* W14, W15, W16, W17 *)
  [ %MF298 := ( ( ( %MF295 + %MF232 ) + %MF235 ) + %MF238 ) + %MF241 ](* W18, W19, W20, W21 *)
  [ %MF301 := ( ( ( %MF298 + %MF244 ) + %MF247 ) + %MF250 ) + %MF253 ](* DEN, W22, W23, W24, W25 *)
  // as ST:
  //   %MF286 := ( ( ( W1 + W2 ) + W3 ) + W4 ) + W5;
  //   %MF289 := ( ( ( %MF286 + W6 ) + W7 ) + W8 ) + W9;
  //   %MF292 := ( ( ( %MF289 + W10 ) + W11 ) + W12 ) + W13;
  //   %MF295 := ( ( ( %MF292 + W14 ) + W15 ) + W16 ) + W17;
  //   %MF298 := ( ( ( %MF295 + W18 ) + W19 ) + W20 ) + W21;
  //   DEN := ( ( ( %MF298 + W22 ) + W23 ) + W24 ) + W25;

// Rung 73: crisp
  LD %I0.0
  [ %MW503 := REAL_TO_INT ( %MF283 / %MF301 ) ](* CRISP, NUM, DEN *)
  // as ST:
  //   IF %I0.0 THEN CRISP := REAL_TO_INT ( NUM / DEN ); END_IF;
